PROGRAM Main
VAR
	task : Task;
	
	axis1 : Axis;	
	
	enable: BOOL;
	disable: BOOL;
	reset: BOOL;
	halt: BOOL;
	stop: BOOL;
	
	startHoming : BOOL;
	homePosition : LREAL := 10;
	homeCam : BOOL;
	
	setPositionAbsolute : BOOL;
	setPositionRelative : BOOL;
	setPositionValue : LREAL;

	jogForward : BOOL;
	jogBackwards : BOOL;
	
	startMove1 : BOOL;
	startMove2 : BOOL;	
	moveVelocity : LREAL := 200;
	movePosition1 : LREAL := 1000;
	movePosition2 : LREAL := 0;
	
	homingFeedback : I_CommandFeedback;
	setPositionFeedback : I_CommandFeedback;
	resetFeedback : I_CommandFeedback;
	haltFeedback : I_CommandFeedback;
	stopFeedback : I_CommandFeedback;
	feedback : I_CommandFeedback;
	feedback2 : I_CommandFeedback;
	
	feedbackToDisplay : I_CommandFeedback;
	fbBusy : BOOL;
	fbDone : BOOL;
	fbError: BOOL;
	fbErrorId: UDINT;
	fbAborting: BOOL;
	fbAborted: BOOL;
	
	isStatusValid: BOOL;
	isAtStandStill: BOOL;
	isAccelerating: BOOL;
	isAtConstantVelocity: BOOL;
	isDecelerating: BOOL;
	isStopping: BOOL;	
	isInContinuousMotion: BOOL;
	isInDiscreteMotion: BOOL;
	isInSynchronizedMotion: BOOL;
	isErrorStopped: BOOL;
	hasError: BOOL;
	errorId: UDINT;
END_VAR

task.CyclicCall();
IF enable THEN
	enable := FALSE;
	axis1.Enable(AxisBufferMode.Buffered);
	axis1.EnablePositive();
	axis1.EnableNegative();
END_IF
IF disable THEN
	disable := FALSE;
	axis1.Disable();
END_IF
IF reset THEN
	reset := FALSE;
	axis1.Reset(resetFeedback);
END_IF
IF halt THEN
	halt := FALSE;
	axis1.Halt(haltFeedback);
END_IF
IF stop THEN
	stop := FALSE;
	axis1.Stop(stopFeedback);
END_IF
IF jogForward THEN
	axis1.JogForward(100);
ELSIF jogBackwards THEN
	axis1.JogBackwards(100);
ELSE
	// Don't like this, since jogging now acts like MC_MoveVelocity
	// although I guess that is what it is exactly
	axis1.StopJogging();
END_IF

IF startHoming THEN
	startHoming := FALSE;
	(*axis1.HomingBuilder()
		.Position(homePosition)
		.BuildDirectHomingCommand()
		.Execute(homingFeedback)
		.ThenRelease();*)
	axis1.HomingBuilder()
		.Position(homePosition)
		.Cam(homeCam)
		.ReferenceMode(EncoderReferenceMode.PLCCam)
		.BuildDefaultHomingCommand()
		.Execute(homingFeedback)
		.ThenRelease();
END_IF

IF setPositionAbsolute THEN
	setPositionAbsolute := FALSE;
	axis1.SetPositionAbsolute(setPositionValue, setPositionFeedback);
END_IF

IF setPositionRelative THEN
	setPositionRelative := FALSE;
	axis1.SetPositionRelative(setPositionValue, setPositionFeedback);
END_IF

IF startMove1 THEN
	startMove1 := FALSE;
	axis1.MoveBuilder()
		.Velocity(100)
		.BufferMode(AxisBufferMode.Aborting)
		.Position(movePosition1)
		.BuildMoveAbsoluteCommand()
		.Execute(feedback)
		.ThenRelease();
END_IF

IF startMove2 THEN
	startMove2 := FALSE;
	axis1.MoveBuilder()
		.Velocity(100)
		.BufferMode(AxisBufferMode.Buffered)
		.Position(movePosition2)
		.BuildMoveAbsoluteCommand()
		.Execute(feedback)
		.ThenRelease();
END_IF

feedbackToDisplay := homingFeedback;
IF feedbackToDisplay <> 0 THEN
	fbBusy := feedbackToDisplay.Busy;
	fbDone := feedbackToDisplay.Done;
	fbError := feedbackToDisplay.Error;
	fbErrorId := feedbackToDisplay.ErrorId;
	fbAborting := feedbackToDisplay.Aborting;
	fbAborted := feedbackToDisplay.Aborted;
END_IF

isStatusValid := axis1.IsStatusValid;
IF axis1.IsStatusValid THEN
	isAtStandStill := axis1.IsAtStandStill;
	isAccelerating := axis1.IsAccelerating;
	isAtConstantVelocity := axis1.IsAtConstantVelocity;
	isDecelerating := axis1.IsDecelerating;
	isStopping := axis1.IsStopping;	
	isInContinuousMotion := axis1.IsInContinuousMotion;
	isInDiscreteMotion := axis1.IsInDiscreteMotion;
	isInSynchronizedMotion := axis1.IsInSynchronizedMotion;
	isErrorStopped := axis1.IsErrorStopped;
	hasError := axis1.HasError;
	errorId := axis1.ErrorId;
END_IF

END_PROGRAM

(* stored: Version 1.1.0.1, ProductVersion 3.1.4024.12
   POU Main: Id {2e61a8d4-f677-443a-9a2d-e2cd0bfcaaea}, SpecialFunc None *)
